(* IEC 61131-3 sources: AXOpen/src/_test/app/src, 3 files *)

(* ---- TestContext.st ---- *)
USING AXOpen.Core;
USING AXOpen.Logging;
USING AXOpen.Messaging;
USING AXOpen.Messaging.Static;

// ============================================================
// TestContext — Documentation AxoContext for the test app.
// Contains documentation examples and core objects.
// Sandbox/testing objects have been moved to src/sandbox/app.
// ============================================================

{S7.extern=ReadWrite}
CLASS TestContext EXTENDS AXOpen.Core.AxoContext
    VAR PUBLIC
        // ---- Components.Rexroth.Drives ----
        rexroth_drives_documentation : AXOpen.Components.Rexroth.Drives.RexrothDrives;

    END_VAR

    METHOD PROTECTED OVERRIDE Main
        THIS.InitializeRootObject(rexroth_drives_documentation);
        rexroth_drives_documentation.Execute();

    END_METHOD
END_CLASS

(* ---- configuration.st ---- *)
USING AXOpen.Core;

// ============================================================
// Showcase unified configuration
// Includes representative examples from every library.
//
// Variable naming convention:
//   - Core / Data / Foundation-lib examples keep their
//     original names where those names are globally unique.
//   - Component-library sandbox/documentation contexts are
//     prefixed with the short library name to avoid conflicts,
//     because each library defines types of the same name in
//     its own namespace.
// ============================================================

CONFIGURATION MyConfiguration
    TASK Main(Interval := T#10ms, Priority := 1);
    PROGRAM P1 WITH Main: TestProgram;

    VAR_GLOBAL
        // ---- Shared RTC / RTM ----
        {S7.extern=ReadWrite}
        _rtc : AXOpen.S71500.Rtc;
        {S7.extern=ReadWrite}
        _rtm : AXOpen.S71500.Rtm;

        // ---- PLC alive counter ----
        {#ix-set:AttributeName = "PLC alive counter"}
        {S7.extern=ReadWrite}
        I_am_alive : ULINT;

        // ---- Single unified context ----
        {S7.extern=ReadWrite}
        Ctx : TestContext;
    END_VAR
END_CONFIGURATION

(* ---- program.st ---- *)
USING AXOpen.Core;

PROGRAM TestProgram
    VAR_EXTERNAL
        _rtc : AXOpen.S71500.Rtc;
        _rtm : AXOpen.S71500.Rtm;
        {#ix-set:AttributeName = "PLC alive counter"}
        I_am_alive : ULINT;
        Ctx : TestContext;
    END_VAR

    I_am_alive := I_am_alive + ULINT#1;

    // Inject shared services into the single unified context
    Ctx.InjectRtc(_rtc);
    Ctx.InjectRtm(_rtm);

    // Run the single context — orchestrates all examples
    Ctx.Run();
END_PROGRAM
